ABB RobotStudio station: Estacion_ABB_AR.rsstn

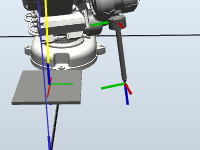
Station Station (saved by RobotStudio 6.8.8148.134)
Controller SistemaTCP, task T_ROB1: task frame (RAPID world) sits at (-700, 0, 0) mm in the station
Controller SistemaTCP
  mechanical unit ROB_1: IRB140_6_81_C_03, 6 joints, base frame (0, 0, 0) mm
Layout (positions relative to the parent item):
  - IRB140_6_81_C_03 [mechanism, from Robots\IRB140_6_81_C_G_03.rslib] at (-700, 0, 0) mm; joint values [0.3069, 0.6939, -0.3021, 0.1347, 1.0865, 3.2301] (rad or m)
  - Tool_Sonda [mechanism] at (-75.42, 206.04, 419.37) mm, rotated rx -172.42 ry -4.42 rz 8.94 deg
      TCP Tool_Sonda_TPC at (0, 0, 200) mm
      links: P_sonda
  - Pieza_1 [part] at (-200, -100, 190) mm
  - Pieza_3 [part]
Attachment: Tool_Sonda is attached to IRB140_6_81_C_03 / Link6
Targets, tools, work objects and paths stored in the station, written as RAPID:
! task T_ROB1
MODULE CalibData
  PERS tooldata Tool_Sonda_TPC:=[TRUE,[[0,0,200],[1,0,0,0]],[0.1,[0,0,1],[1,0,0,0],0,0,0]];
  TASK PERS wobjdata Wobj_Origen_unal:=[FALSE,TRUE,"",[[600,0,200],[1,0,0,0]],[[0,0,0],[1,0,0,0]]];
  CONST robtarget HOME:=[[506.291626224,0,679.694493073],[0.499999994,0,0.866025407,0],[0,0,0,0],[9E+09,9E+09,9E+09,9E+09,9E+09,9E+09]];
ENDMODULE

! task T_ROB1
MODULE Module1
  CONST robtarget Cuadro1:=[[679.496708571,159.713796026,452.928593845],[0.500000008,0.000000022,0.866025399,0.000000005],[0,-1,0,0],[9E+09,9E+09,9E+09,9E+09,9E+09,9E+09]];
  CONST robtarget Cuadro2:=[[679.496707444,159.713813829,591.47851807],[0.500000012,0.000000025,0.866025397,0.000000014],[0,-1,0,0],[9E+09,9E+09,9E+09,9E+09,9E+09,9E+09]];
  CONST robtarget Cuadro3:=[[679.496709501,-236.924493196,591.478513946],[0.500000009,0.000000027,0.866025398,0.000000022],[-1,0,-1,0],[9E+09,9E+09,9E+09,9E+09,9E+09,9E+09]];
  CONST robtarget Cuadro4:=[[679.496706459,-236.924493019,441.939874989],[0.5,-0.000000009,0.866025404,0.000000001],[-1,0,-1,0],[9E+09,9E+09,9E+09,9E+09,9E+09,9E+09]];
  PROC Path_10()
  ENDPROC
ENDMODULE

! task T_ROB1
MODULE MOD1
  PROC main()
    MoveL HOME,v400,z100,tool0\WObj:=wobj0;
    WaitTime 4;
    MoveL il_1,v1000,fine,Tool_Sonda_TPC\WObj:=Wobj_Origen_unal;
    WaitTime 2;
  ENDPROC
ENDMODULE

